{attribute addProperty BoxType "EJ6002-0000-0016"}
{attribute addProperty Id "COM_Inputs_ChannelAT %I*ARRAY[0..1] OF COM_Inputs_Channel_85D1D733384480COM_Outputs_ChannelAT %Q*ARRAY[0..1] OF COM_Outputs_Channel_85BCA431384480WcStateAT %I*WcState_F855686C1620InfoDataAT %I*InfoData_BC63D37F80100"}
{attribute addProperty CRC "60965666"}
{attribute addProperty SizeInBites "864"}
{attribute addProperty SizeInBytes "108"}
TYPE EJ6002_A0C112E7 :
STRUCT
	{attribute addProperty Name "COM_Inputs_Channel"}
	COM_Inputs_Channel : ARRAY[0..1] OF COM_Inputs_Channel_85D1D733;
	{attribute addProperty Name "COM_Outputs_Channel"}
	COM_Outputs_Channel : ARRAY[0..1] OF COM_Outputs_Channel_85BCA431;
	{attribute addProperty Name "WcState"}
	WcState : WcState_F855686C;
	{attribute addProperty Name "InfoData"}
	InfoData : InfoData_BC63D37F;
END_STRUCT
END_TYPE

(* stored: Version 1.2.0.0, ProductVersion 3.1.4024.9
   DUT EJ6002_A0C112E7: Id {8dd82e56-8265-4c2a-9870-a36018c0429f} *)
